// TwinCAT 3 PLC project Plc
// ProgramVersion: 3.1.4024.0
// libraries:
//   Tc2_Standard, * (Beckhoff Automation GmbH)
//   Tc2_System, * (Beckhoff Automation GmbH)
//   Tc3_Module, * (Beckhoff Automation GmbH)
//   VisuSymbols,3.5.10.0,System
// project tree:
//   / Gestore di visualizzazione.TcVMO (not stored), GlobalTextList.TcGTLO, PlcTask.TcTTO
//   GVLs/ GVL.TcGVL
//   POUs/ MAIN.TcPOU
//   VISUs/ Visualization.TcVIS
// real-time tasks:
//   TASK PlcTask: cycle T#10ms, priority 20, ADS port 350

CONFIGURATION Plc
    RESOURCE PLC ON TwinCAT3
        TASK PlcTask(INTERVAL := T#10ms, PRIORITY := 20);
        PROGRAM MAIN WITH PlcTask : MAIN;
    END_RESOURCE
END_CONFIGURATION

// ---- GVLs/GVL.TcGVL
{attribute 'qualified_only'}
VAR_GLOBAL
	pBDelay: BOOL;
	probeDelay: BOOL;
	pbTimer: BOOL;
	probeTimer: BOOL;
	pbBlink: BOOL;
	blinkEnable: BOOL;
	probeBlink: BOOL;
	pbClear: BOOL;
END_VAR

// ---- POUs/MAIN.TcPOU
PROGRAM MAIN
VAR
	TONDelay: TON;
	TONTimer: TON;
	TONBlink1: TON;
	TONBlink2: TON;
END_VAR

Delay();
Timer();
Blink();

ACTION Blink:
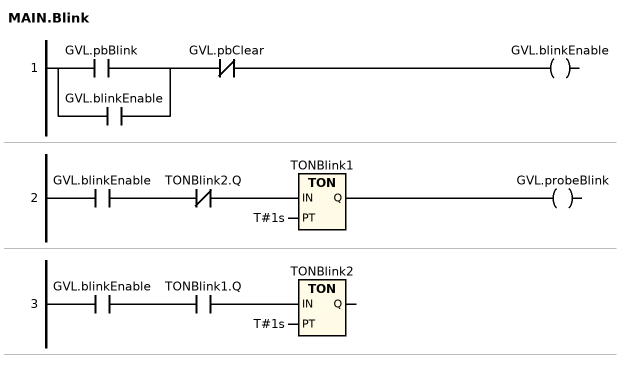
// NETWORK 1
GVL.blinkEnable := (GVL.pbBlink OR GVL.blinkEnable) AND NOT GVL.pbClear;

// NETWORK 2
TONBlink1(IN := GVL.blinkEnable AND NOT TONBlink2.Q, PT := T#1s); // TON
GVL.probeBlink := TONBlink1.Q;

// NETWORK 3
TONBlink2(IN := GVL.blinkEnable AND TONBlink1.Q, PT := T#1s); // TON
END_ACTION

ACTION Delay:
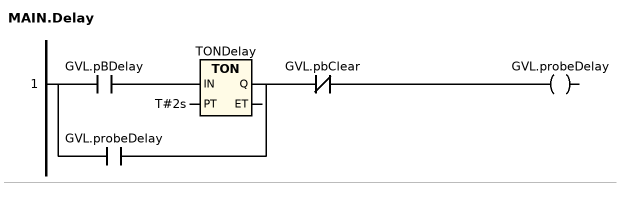
// NETWORK 1
TONDelay(IN := GVL.pBDelay, PT := T#2s); // TON
GVL.probeDelay := (TONDelay.Q OR GVL.probeDelay) AND NOT GVL.pbClear;
END_ACTION

ACTION Timer:
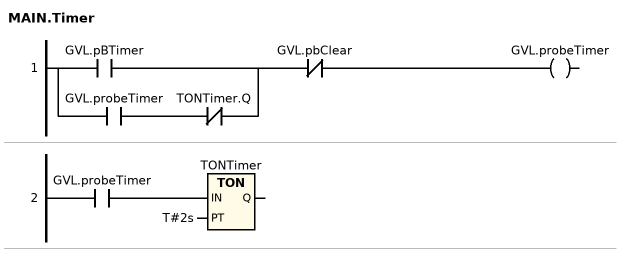
// NETWORK 1
GVL.probeTimer := (GVL.pBTimer OR GVL.probeTimer AND NOT TONTimer.Q) AND NOT GVL.pbClear;

// NETWORK 2
TONTimer(IN := GVL.probeTimer, PT := T#2s); // TON
END_ACTION

END_PROGRAM

// ---- GlobalTextList.TcGTLO
TEXTLIST GlobalTextList
  107 = 'Blink'
  196 = 'Clear'
  191 = 'Delay'
  662 = 'Timer'
END_TEXTLIST

// ---- VISUs/Visualization.TcVIS
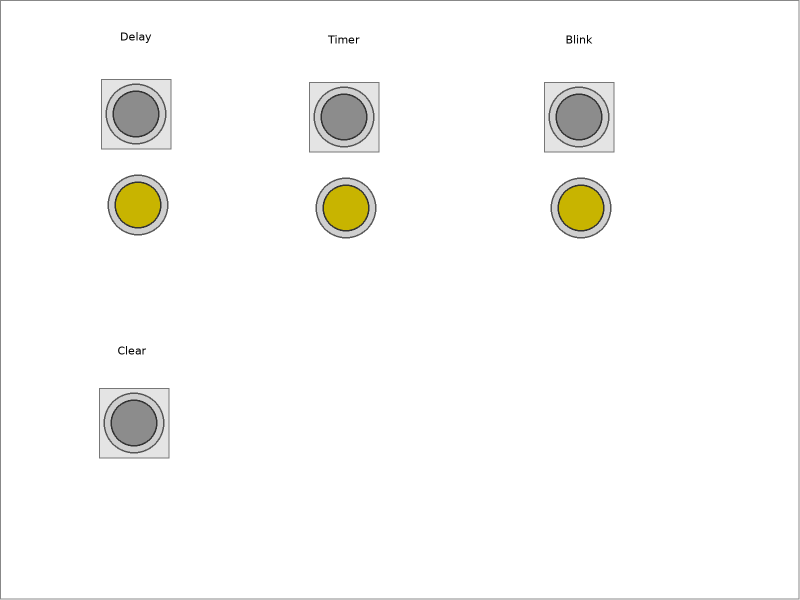
VISUALIZATION Visualization  // 800x600
    Lamp1 (103,170 70x70), variable: GVL.probeDelay, style: Lamp-Lamp1-Yellow
    PushSwitch (101,79 70x70), variable: GVL.pBDelay, behaviour: TAP, style: Switch-PushSwitch-Gray
    Label (61,22 150x30), "Delay"
    PushSwitch (99,388 70x70), variable: GVL.pbClear, behaviour: TAP, style: Switch-PushSwitch-Gray
    Label (57,336 150x30), "Clear"
    Lamp1 (311,173 70x70), variable: GVL.probeTimer, style: Lamp-Lamp1-Yellow
    PushSwitch (309,82 70x70), variable: GVL.pbTimer, behaviour: TAP, style: Switch-PushSwitch-Gray
    Label (269,25 150x30), "Timer"
    Lamp1 (546,173 70x70), variable: GVL.probeBlink, style: Lamp-Lamp1-Yellow
    PushSwitch (544,82 70x70), variable: GVL.pbBlink, behaviour: TAP, style: Switch-PushSwitch-Gray
    Label (504,25 150x30), "Blink"
END_VISUALIZATION
